GLOBALCONSTANTS myComputers (* Global constants *)
  (* Standard: 61499-1; Description: Copyright (c) 2023 HR Agrartechnik GmbH This program and the accompanying materials are made available under the terms of the Eclipse Public License 2.0 which is available at https://www.eclipse.org/legal/epl-2.0/ SPDX-License-Identifier: EPL-2.0 *)
  (* Version 1.0, 2023-10-22, Franz Höpfinger, HR Agrartechnik GmbH *)
  PACKAGE VV::const::Computers;
  VAR_GLOBAL CONSTANT
    C_PC_SERVER : WSTRING := "192.168.178.126:61499";
    C_PC_CLIENT : WSTRING := "192.168.178.127:61499";
    C_PC_PUBLISH : WSTRING := "192.168.178.60:61499";
    C_PC_SUBSCRIBE : WSTRING := "192.168.178.62:61499";
  END_VAR
END_GLOBALCONSTANTS
